Fanuc KAREL source: kb00167.KL

-- PROVISIONAL review KL for V770-1; original PC SHA256 a70121cfb5a13634227e796497acebca11e24c2c075e5881c30e1cd8784e939f
-- Incomplete behavior may be omitted. Consult companion uncertainty JSON. Do not deploy.
PROGRAM KB00167
%NOLOCKGROUP
BEGIN
  -- UNRESOLVED_PC offsets 5-12; opcodes 9D,23
  -- UNRESOLVED_PC offsets 17-24; opcodes 9D,23
  -- UNRESOLVED_PC offsets 29-36; opcodes 9D,23
  -- UNRESOLVED_PC offsets 41-77; opcodes 27,22,22,22,1C,22,27,9D,31
  -- UNRESOLVED_PC offsets 82-86; opcodes 7F
END KB00167
